// TwinCAT 3 PLC project IBF_HMI
// Title: IBF_HMI
// Company: Industrial Brains B.V.
// ProjectVersion: 0.0.0.0
// Description: Basic HMI screens for use with Utilities and device libraries
// ProgramVersion: 3.1.4023.0
// libraries:
//   IBF_Devices, * (Industrial Brains B.V.)
//   IBF_Utilities, * (Industrial Brains B.V.)
//   Tc2_Standard, * (Beckhoff Automation GmbH)
//   Tc2_System, * (Beckhoff Automation GmbH)
//   Tc2_Utilities, * (Beckhoff Automation GmbH)
//   Tc3_Module, * (Beckhoff Automation GmbH)
//   VisuDialogs, * (System)
//   VisuSymbols,3.5.10.0,System
// project tree:
//   HMIControl/DataTypes/ E_BaseVisu.TcTLEO, UDT_HMI_FaultLogItem.TcDUT, UDT_HMI_LogItem.TcDUT
//   HMIControl/ FB_LogView.TcPOU, FB_HMIControl.TcPOU
//   IconsAndPictures/Backgrounds/ BackgroundImagePool_PNG.TcIPO (not stored), BackGroundImagePool_SVG.TcIPO (not stored)
//   / PlcTask.TcTTO, VisualizationManager.TcVMO (not stored), VISU_TASK.TcTTO
//   Screens/Backgrounds/ BG_Borders.TcVIS, BG_Emergency.TcVIS, BG_Logo_IndustrialBrains.TcVIS
//   Screens/Base/ BaseScreen.TcVIS
//   Screens/Buttons/ ButtonHome.TcVIS, ButtonLogin.TcVIS, ButtonManual.TcVIS, ButtonSettings.TcVIS, ButtonParameters.TcVIS, ButtonLog.TcVIS, ButtonTemplate.TcVIS
//   Screens/LogView/ LogView.TcVIS
//   Screens/Parameter/ ParameterControl.TcVIS
//   Screens/State/ Idle.TcVIS, Manual.TcVIS, Parameters.TcVIS, FaultLog.TcVIS
//   Tools/Colors/ E_Color.TcDUT, F_GetColor.TcPOU, F_GetTransparantColor.TcPOU, U_Color.TcDUT
//   Tools/InputFunctions/ FB_HMIInputBase.TcPOU, FB_HMILREALInput.TcPOU
//   _TESTS/ FB_Base_Test.TcPOU, PRG_TEST.TcPOU, PRG_TEST_GLOBAL.TcPOU, PRG_TEST_LOGVIEW.TcPOU, VISU_DummyState.TcVIS, VISU_TEST_BASE.TcVIS, VISU_TEST_LOGVIEW.TcVIS
//   GVL/ GVL_HMI.TcGVL
//   IconsAndPictures/Buttons/ Buttons_SVG.TcIPO (not stored), Buttons_PNG.TcIPO (not stored)
//   IconsAndPictures/Logos/ LogoPool.TcIPO (not stored)
//   TextLists/ E_ComponentTypes.TcTLO, E_FaultTypes.TcTLO (not stored), E_Locations.TcTLO (not stored), E_MessageNumbers.TcTLO, E_ParameterNames.TcTLO (not stored), GlobalTextList.TcGTLO, TL_MessageDiscriptions.TcTLO (not stored)
// real-time tasks:
//   TASK PlcTask: cycle T#10ms, priority 6, ADS port 350
//   TASK VISU_TASK: cycle T#100000us, priority 8, ADS port 351

CONFIGURATION IBF_HMI
    RESOURCE PLC ON TwinCAT3
        TASK PlcTask(INTERVAL := T#10ms, PRIORITY := 6);
        TASK VISU_TASK(INTERVAL := T#100000us, PRIORITY := 8);
        PROGRAM PRG_TEST_GLOBAL WITH PlcTask : PRG_TEST_GLOBAL;
        PROGRAM PRG_TEST WITH PlcTask : PRG_TEST;
        PROGRAM PRG_TEST_LOGVIEW WITH PlcTask : PRG_TEST_LOGVIEW;
        PROGRAM VisuElems_Visu_Prg WITH VISU_TASK : VisuElems.Visu_Prg;
    END_RESOURCE
END_CONFIGURATION

// ---- HMIControl/DataTypes/E_BaseVisu.TcTLEO
{attribute 'qualified_only'}
{attribute 'strict'}
TYPE E_BaseVisu :
(
	Idle := 0,
	Settings,
	Parameter,
	Manual,
	SemiAutomatic,
	Automatic,
	LogView
)INT;
END_TYPE

// ---- HMIControl/DataTypes/UDT_HMI_FaultLogItem.TcDUT
TYPE UDT_HMI_FaultLogItem :
STRUCT
	sID : STRING;
	sDescription : STRING;
	sStartTime : STRING[19];
	sEndTime : STRING[19];
	dColor_Bg : DWORD := E_Color.White; // Table row background color
END_STRUCT
END_TYPE

// ---- HMIControl/DataTypes/UDT_HMI_LogItem.TcDUT
TYPE UDT_HMI_LogItem :
STRUCT
	sTimestamp : STRING[23];
	sLevel : STRING;
	sMsg : T_MaxString;
	dColor_Bg : DWORD := E_Color.White; // Table row background color
END_STRUCT
END_TYPE

// ---- Tools/Colors/E_Color.TcDUT
{attribute 'qualified_only'}
{attribute 'strict'}
TYPE E_Color : // Theme colors
(
	Bg_Light	:= 16#FF19A9E1, // Theme background color (light blue)
	Bg_Dark		:= 16#FF122941, // Theme background color (dark blue)

	White 		:= 16#FFFFFFFF,
	Black 		:= 16#FF000000,

	DarkRed		:= 16#FFFF0000,
	LightRed	:= 16#FFFF8888,
	DarkYellow 	:= 16#FFFFFF00,
	LightYellow := 16#FFFFFF88,
	DarkGreen 	:= 16#FF00FF00,
	LightGreen	:= 16#FF88FF88

) DWORD;
END_TYPE

// ---- Tools/Colors/U_Color.TcDUT
TYPE U_Color :
UNION
	rgba : ARRAY[0..3] OF BYTE;
	dw : DWORD;
END_UNION
END_TYPE

// ---- GVL/GVL_HMI.TcGVL
{attribute 'qualified_only'}
VAR_GLOBAL
	fbHMIControl	: FB_HMIControl ; // HMI control function
END_VAR

// ---- _TESTS/PRG_TEST_GLOBAL.TcPOU
PROGRAM INTERNAL PRG_TEST_GLOBAL // A place to call global function blocks (singletons) that can be used by all tests

Sys_Variables.fbSystemVariables();
GVL_Utilities.fbFaultHandler();

END_PROGRAM

// ---- _TESTS/PRG_TEST.TcPOU
PROGRAM INTERNAL PRG_TEST
VAR
	fbLogHandler_PersistentArray : FB_LogHandler_PersistentArray;
	bInitDone 	: BOOL;
	fbDevValve 	: FB_DevValve;
END_VAR

// NOTE: fbParameterHandler should contain the parameters of fbDevValve. 
// Parameter values are persistent
IF NOT bInitDone THEN
	bInitDone := TRUE;
	fbDevValve.Init(
		nId := 1,
		nParentId := 0,
		eResetState := E_ValveResetState.Res_Idle,
		eSafeState := E_ValveResetState.Res_Idle
	);
END_IF

fbDevValve();

GVL_Parameters.fbParameterHandler();

GVL_HMI.fbHMIControl(fbLogHandler_PersistentArray := fbLogHandler_PersistentArray);

END_PROGRAM

// ---- _TESTS/PRG_TEST_LOGVIEW.TcPOU
PROGRAM INTERNAL PRG_TEST_LOGVIEW
VAR
	fbLogHandler_PersistentArray : FB_LogHandler_PersistentArray;
	bEnableTests : BOOL;
	fbLogView : FB_LogView;
	fbLogger : FB_Logger;
	fbBase : FB_Base_Test;
	bCmdReset : BOOL;
END_VAR

IF bEnableTests THEN

	fbLogView(fbLogHandler_PersistentArray := fbLogHandler_PersistentArray);

	fbBase();

	IF bCmdReset THEN
		bCmdReset R= GVL_Utilities.fbFaultHandler.CmdReset();
	END_IF
	
END_IF

END_PROGRAM

// ---- HMIControl/FB_LogView.TcPOU
FUNCTION_BLOCK INTERNAL FB_LogView
VAR CONSTANT
	NUMBER_OF_ITEMS_IN_TABLE : UINT := 16;
END_VAR
VAR_INPUT
	bAcknowledge : BOOL; // Clear inactive items from the log
	bReset : BOOL; // Reset faults
	bBlinkButton : BOOL; // Blink the button to alert operator (optional, not used thusfar)
	fbLogHandler_RetainableList : REFERENCE TO FB_LogHandler_RetainableList; // Optional reference to a FB_LogHandler_RetainableList instance
END_VAR
VAR_OUTPUT
	arLog : ARRAY[1..NUMBER_OF_ITEMS_IN_TABLE] OF UDT_HMI_FaultLogItem;
	arHistory : ARRAY[1..GVL_Utilities.RETAINABLE_LOG_HISTORY_SIZE] OF UDT_HMI_LogItem;
	
	// Log button properties
	dLogButtonColor 	: DWORD;
	nLogButtonNumber 	: UINT;
		
	reNewLogMessages : BOOL; // TRUE when new log messages arrive (for one cycle)
	nPrevFaultsInLog : UINT;
END_VAR
VAR
	fbFormatString : FB_FormatString;
END_VAR
VAR_TEMP
	i : UINT; // Iterator
	nArHistoryIndex : UINT; // arHistory array index
	
	stLogItem : UDT_LogItem;
	stFaultLogItem : UDT_FaultLogItem;
	stEmptyFaultLogItem : UDT_HMI_FaultLogItem;
	
	fMonth : REAL;
	fDay : REAL;
	fHour : REAL;
	fMinute : REAL;
	fSecond : REAL;
	fMilliseconds : REAL;	
END_VAR

{region 'FAULT LOG / ALARM BELL ICON'}
// Report new log messages
reNewLogMessages := (GVL_Utilities.fbFaultHandler.nFaultsInLog > nPrevFaultsInLog);
nPrevFaultsInLog := GVL_Utilities.fbFaultHandler.nFaultsInLog;

// Update array
stFaultLogItem := GVL_Utilities.fbFaultHandler.Head;
FOR i := 1 TO NUMBER_OF_ITEMS_IN_TABLE DO
	IF i <= GVL_Utilities.fbFaultHandler.nFaultsInLog THEN
		arLog[i].sID := stFaultLogItem.Id;
		arLog[i].sDescription := stFaultLogItem.stFault.Description;
		arLog[i].sStartTime := DT_To_Str(stFaultLogItem.StartTime);
		arLog[i].sEndTime := DT_To_Str(stFaultLogItem.EndTime);
		IF stFaultLogItem.stFault.Active THEN
			arLog[i].dColor_Bg := GetFaultTypeColorBG(stFaultLogItem.stFault.FaultType);
		ELSE
			arLog[i].dColor_Bg := E_Color.White;
		END_IF
		stFaultLogItem := GVL_Utilities.fbFaultHandler.Next;
	ELSE
		arLog[i] := stEmptyFaultLogItem;
	END_IF
END_FOR

// Set log button properties
nLogButtonNumber := GVL_Utilities.fbFaultHandler.nFaultsInLog;
// Set color, in order of priority
IF bBlinkButton AND Sys_Variables.BlinkFast THEN
	dLogButtonColor := E_Color.Bg_Dark;
ELSIF GVL_Utilities.fbFaultHandler.arActiveFaultTypes[E_FaultTypes.FF] THEN
	dLogButtonColor := GetFaultTypeColorBG(E_FaultTypes.FF);
ELSIF GVL_Utilities.fbFaultHandler.arActiveFaultTypes[E_FaultTypes.CF] THEN
	dLogButtonColor := GetFaultTypeColorBG(E_FaultTypes.CF);
ELSIF GVL_Utilities.fbFaultHandler.arActiveFaultTypes[E_FaultTypes.MC] THEN
	dLogButtonColor := GetFaultTypeColorBG(E_FaultTypes.MC);
ELSIF GVL_Utilities.fbFaultHandler.arActiveFaultTypes[E_FaultTypes.OW] THEN
	dLogButtonColor := GetFaultTypeColorBG(E_FaultTypes.OW);
ELSIF GVL_Utilities.fbFaultHandler.arActiveFaultTypes[E_FaultTypes.OM] THEN
	dLogButtonColor := GetFaultTypeColorBG(E_FaultTypes.OM);
ELSE
	dLogButtonColor := E_Color.Bg_Light;
END_IF 

IF bAcknowledge THEN
	bAcknowledge R= GVL_Utilities.fbFaultHandler.CmdClearInactive();
END_IF

IF bReset THEN
	bReset R= GVL_Utilities.fbFaultHandler.CmdReset();
END_IF
{endregion}

{region 'Log history'}
IF __ISVALIDREF(fbLogHandler_RetainableList) THEN
	// Add items from retainable list in reversed order, starting with the last added item
	nArHistoryIndex := 0;
	FOR i := (fbLogHandler_RetainableList.nIndex + GVL_Utilities.RETAINABLE_LOG_HISTORY_SIZE - 1) TO fbLogHandler_RetainableList.nIndex BY -1 DO
		nArHistoryIndex := nArHistoryIndex + 1;
		stLogItem := fbLogHandler_RetainableList.aLogItems[(i MOD GVL_Utilities.RETAINABLE_LOG_HISTORY_SIZE) + 1];
		arHistory[nArHistoryIndex].sMsg := TO_STRING(stLogItem.sMsg);
		arHistory[nArHistoryIndex].sLevel := TO_STRING(stLogItem.eLevel);
		arHistory[nArHistoryIndex].dColor_Bg := GetLevelColorBG(stLogItem.eLevel);

		// Build timestamp string
		fMonth := WORD_TO_REAL(stLogItem.stTimestamp.wMonth); 
		fDay := WORD_TO_REAL(stLogItem.stTimestamp.wDay); 
		fHour := WORD_TO_REAL(stLogItem.stTimestamp.wHour); 
		fMinute := WORD_TO_REAL(stLogItem.stTimestamp.wMinute); 
		fSecond := WORD_TO_REAL(stLogItem.stTimestamp.wSecond); 
		fMilliseconds := WORD_TO_REAL(stLogItem.stTimestamp.wMilliseconds);
		fbFormatString(
			sFormat := '%u-%02.0f-%02.0f %02.0f:%02.0f:%02.0f.%03.0f',
			arg1 := F_WORD(stLogItem.stTimestamp.wYear),
			arg2 := F_REAL(fMonth),
			arg3 := F_REAL(fDay),
			arg4 := F_REAL(fHour),
			arg5 := F_REAL(fMinute),
			arg6 := F_REAL(fSecond),
			arg7 := F_REAL(fMilliseconds),
			sOut => arHistory[nArHistoryIndex].sTimestamp
		);
	END_FOR
END_IF
{endregion}

METHOD PRIVATE GetFaultTypeColorBG : DWORD
VAR_INPUT
	eFaultType : E_FaultTypes;
END_VAR
CASE eFaultType OF
	E_FaultTypes.FF:
		GetFaultTypeColorBG := E_Color.LightRed;
	E_FaultTypes.CF:
		GetFaultTypeColorBG := E_Color.LightRed;
	E_FaultTypes.MC:
		GetFaultTypeColorBG := E_Color.LightYellow;
	E_FaultTypes.OW:
		GetFaultTypeColorBG := E_Color.LightYellow;
	E_FaultTypes.OM:
		GetFaultTypeColorBG := E_Color.Bg_Light;
END_CASE
END_METHOD

METHOD PRIVATE GetLevelColorBG : DWORD
VAR_INPUT
	eLogLevel : E_LogLevel;
END_VAR
CASE eLogLevel OF
	E_LogLevel.TRACE:
		GetLevelColorBG := E_Color.White;
	E_LogLevel.DEBUG:
		GetLevelColorBG := E_Color.White;
	E_LogLevel.INFO:
		GetLevelColorBG := E_Color.LightGreen;
	E_LogLevel.WARN:
		GetLevelColorBG := E_Color.LightYellow;
	E_LogLevel.ERROR:
		GetLevelColorBG := E_Color.LightRed;
	E_LogLevel.FATAL:
		GetLevelColorBG := E_Color.LightRed;
END_CASE
END_METHOD

END_FUNCTION_BLOCK

// ---- _TESTS/FB_Base_Test.TcPOU
FUNCTION_BLOCK INTERNAL FB_Base_Test EXTENDS FB_Base

SUPER^();

METHOD PUBLIC Init : BOOL
VAR_INPUT
	nId				: UINT ; // Identification number of object
	nParentId		: UINT ; // Id of higher level if applicable (0 = no parent)
	eComponentType	: E_ComponentTypes ; // Component or function type
END_VAR
// Every FB_Base instance is expected to have an Init method that calls ExecIdentifyDevice. 
// This Init method will have at least the nId and nParentId inputs.
// The eComponentType input is optional (can be hardcoded in the Init method, for example see FB_Step).
// It might also have additional inputs (changing the method signature) therefore it is not declared in FB_Base.
ExecIdentifyDevice(nId,	nParentId,	eComponentType);
END_METHOD

END_FUNCTION_BLOCK

// ---- HMIControl/FB_HMIControl.TcPOU
FUNCTION_BLOCK FB_HMIControl
VAR_INPUT
	eScreenRequest 			: E_BaseVisu;
	eHomeScreen   			: E_BaseVisu := E_BaseVisu.Idle; // Home screen is based on system state, e.g., Idle, Automatic, etc.

	bShowEmergencyOverlay 	: BOOL;
	sEmergencyText 			: STRING; // Visible when emergency overlay is shown
	sStatusText 			: STRING; // Text in the bottom border of the screen 

	fbLogHandler_RetainableList : REFERENCE TO FB_LogHandler_RetainableList; // Optional reference to a FB_LogHandler_RetainableList instance
END_VAR
VAR_OUTPUT
	eShownScreen : E_BaseVisu := E_BaseVisu.Idle;

	// Screen states
	bInScreenHome 		: BOOL;
	bInScreenSettings 	: BOOL;
	bInScreenManual 	: BOOL;
	bInScreenParameters	: BOOL;
	bInScreenLog		: BOOL;
	
	// Hide admin/service level navigation buttons
	bHideSecureButtons : BOOL;
END_VAR
VAR
	fbLogView			: FB_LogView;

	feWriteParameter 	: F_TRIG ; // Falling edge trigger on leaving parameter or manual screen
	bWritePar  			: BOOL ; // Busy writing parameters
END_VAR

// Run log view handler
fbLogView(fbLogHandler_RetainableList := fbLogHandler_RetainableList);

// Check user level
bHideSecureButtons := NOT (VisuElems.CurrentUserGroupName = "Admin" OR VisuElems.CurrentUserGroupName = "Service");

// Check if logged in user is allowed to be in the current screen. If not, go to home screen.
IF bHideSecureButtons AND ((eShownScreen = E_BaseVisu.Manual) OR (eShownScreen = E_BaseVisu.Parameter)) THEN
	eScreenRequest := E_BaseVisu.Idle;
END_IF 

// Switch screen
IF (eScreenRequest = E_BaseVisu.Idle) THEN
	eShownScreen := eHomeScreen;
ELSIF (eScreenRequest <> eShownScreen) THEN
	eShownScreen := eScreenRequest;
END_IF

// Report screen states
bInScreenHome 		:= (eShownScreen = eHomeScreen); 
bInScreenSettings 	:= (eShownScreen = E_BaseVisu.Settings);
bInScreenManual 	:= (eShownScreen = E_BaseVisu.Manual);
bInScreenLog 		:= (eShownScreen = E_BaseVisu.LogView);
bInScreenParameters := (eShownScreen = E_BaseVisu.Parameter);

// Save parameters after leaving parameter of manual screen
// Note: in manual operation one can change parameters as well ("learn" function)
feWriteParameter(CLK := (eShownScreen = E_BaseVisu.Parameter) OR (eShownScreen = E_BaseVisu.Manual));
IF feWriteParameter.Q THEN
	bWritePar := TRUE;
END_IF
IF bWritePar THEN 
	bWritePar R= GVL_Parameters.fbParameterHandler.CmdSavePar();
END_IF

END_FUNCTION_BLOCK

// ---- Tools/Colors/F_GetColor.TcPOU
FUNCTION F_GetColor : DWORD // Return an opaque color in DWORD format for use in visualisation
VAR_INPUT
	Red : BYTE;
	Green : BYTE;
	Blue : BYTE;
END_VAR
VAR
END_VAR

F_GetColor := F_GetTransparantColor(Red, Green, Blue, 16#FF);

END_FUNCTION

// ---- Tools/Colors/F_GetTransparantColor.TcPOU
FUNCTION F_GetTransparantColor : DWORD  // Return a transparant color in DWORD format for use in visualisation
VAR_INPUT
	Red : BYTE;
	Green : BYTE;
	Blue : BYTE;
	Alpha : BYTE := 16#FF; // Transparancy, 0 = fully transparant
END_VAR
VAR
	uColor : U_Color;
END_VAR

uColor.rgba[0] := Red;
uColor.rgba[1] := Green;
uColor.rgba[2] := Blue;
uColor.rgba[3] := Alpha;
F_GetTransparantColor := uColor.dw;

END_FUNCTION

// ---- Tools/InputFunctions/FB_HMIInputBase.TcPOU
FUNCTION_BLOCK ABSTRACT FB_HMIInputBase //Base function for HMI inputs
VAR_INPUT
	bEnable : BOOL := TRUE ;
END_VAR
VAR_OUTPUT
	bInVisible			: BOOL := TRUE ; // input is visible (standard := NOT bEnable )
	bDeactivateInput	: BOOL := TRUE ; // input is enabled (Standard := bEnable)
END_VAR
VAR
END_VAR

SetHMIInstructions();

METHOD INTERNAL SetHMIInstructions : BOOL
VAR_INPUT
END_VAR
bInVisible 			:= NOT bEnable ;
bDeactivateInput	:= NOT bEnable ;
END_METHOD

METHOD ABSTRACT SetOutputToPLC : BOOL
VAR_INPUT
END_VAR
END_METHOD

END_FUNCTION_BLOCK

// ---- Tools/InputFunctions/FB_HMILREALInput.TcPOU
FUNCTION_BLOCK PUBLIC FB_HMILREALInput EXTENDS FB_HMIInputBase // Analog value input from HMI
VAR_INPUT
	fInputFromHMI	: LREAL ;
END_VAR
VAR_OUTPUT
	fOutputToPLC	: LREAL ;
END_VAR
VAR
END_VAR

// call base function 
SUPER^();

// Set output to PLC
SetOutputToPLC();

METHOD PUBLIC SetOutputToPLC : BOOL
VAR_INPUT
END_VAR
IF bEnable THEN 
	fOutputToPLC := fInputFromHMI ;
END_IF
END_METHOD

END_FUNCTION_BLOCK

// ---- Screens/Backgrounds/BG_Borders.TcVIS
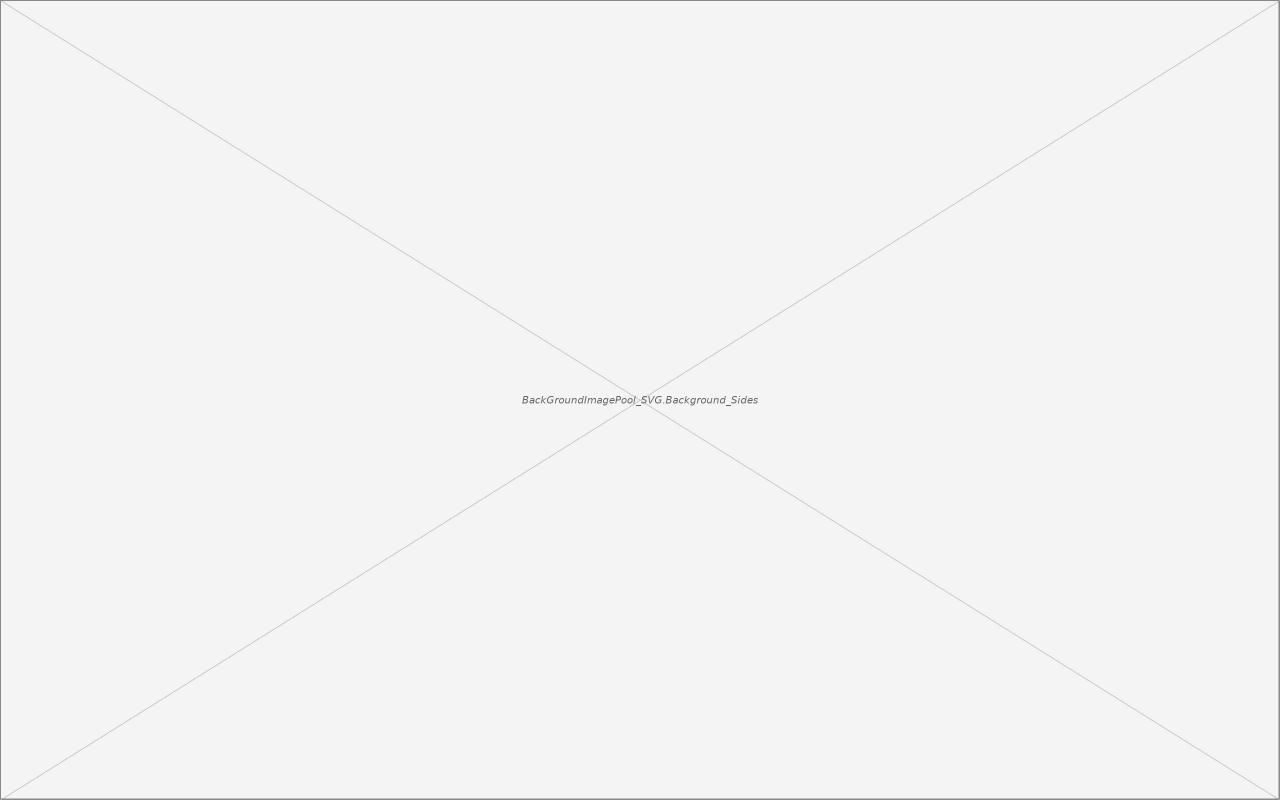
VISUALIZATION BG_Borders  // 1280x800
    Image (0,710 1280x90), image: BackGroundImagePool_SVG.Background_Bottom
    Image (0,0 1280x800), image: BackGroundImagePool_SVG.Background_Sides
END_VISUALIZATION

// ---- Screens/Backgrounds/BG_Emergency.TcVIS
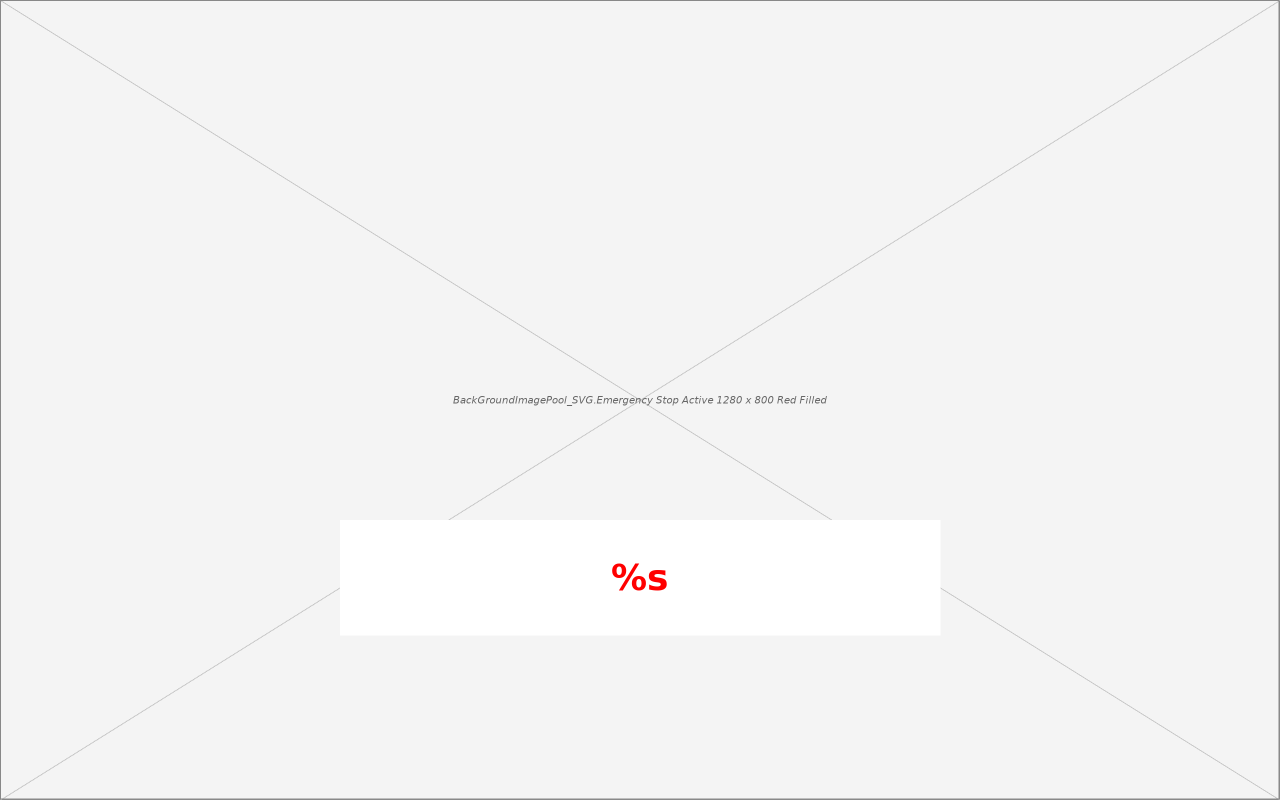
VISUALIZATION BG_Emergency  // 1280x800
VAR_IN_OUT
	sMessage : STRING;
END_VAR
    Image (0,0 1280x800), invisible if: NOT GVL_HMI.fbHMIControl.bShowEmergencyOverlay, image: BackGroundImagePool_SVG.Emergency Stop Active 1280 x 800 Red Filled
    Textfield (340,520 600x115), "%s", text variable: sMessage
END_VISUALIZATION

// ---- Screens/Backgrounds/BG_Logo_IndustrialBrains.TcVIS
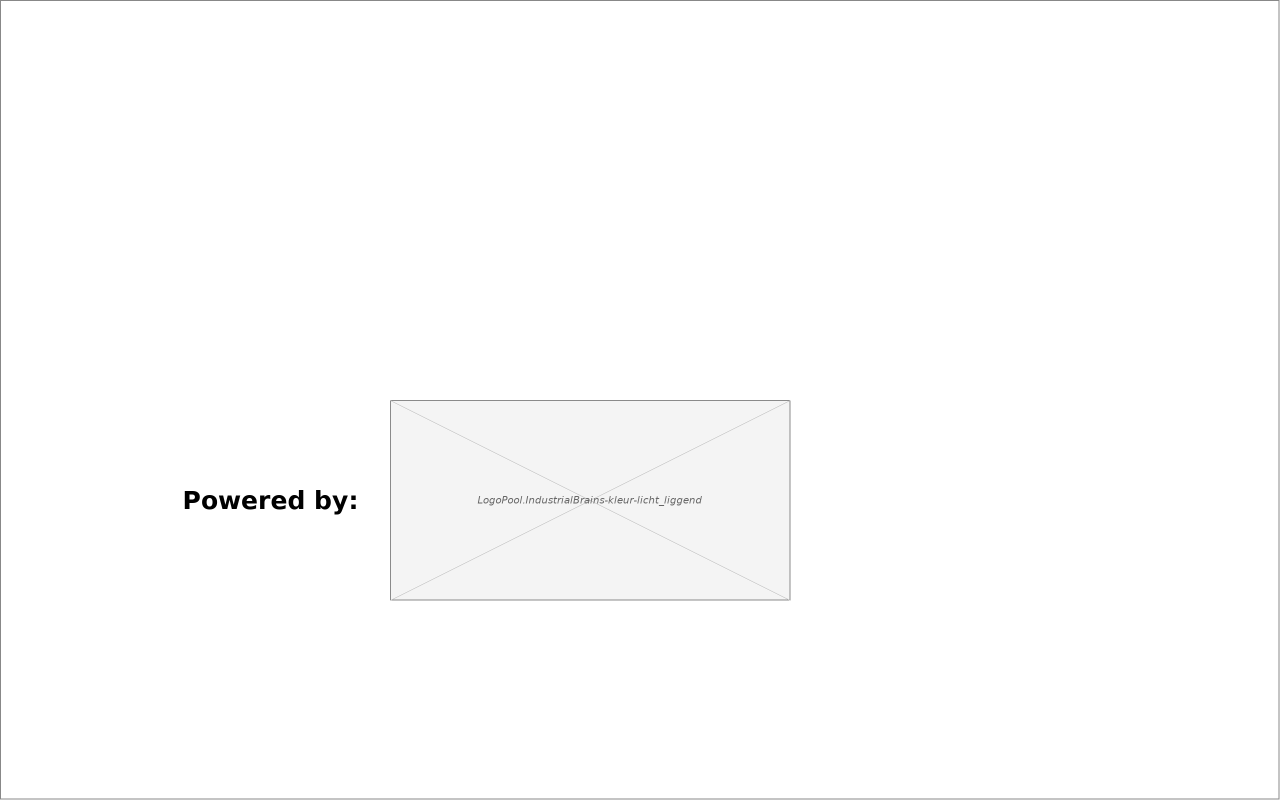
VISUALIZATION BG_Logo_IndustrialBrains  // 1280x800
    Image (390,400 400x200), image: LogoPool.IndustrialBrains-kleur-licht_liggend
    Label (170,400 200x200), "Powered by:"
END_VISUALIZATION

// ---- Screens/Base/BaseScreen.TcVIS
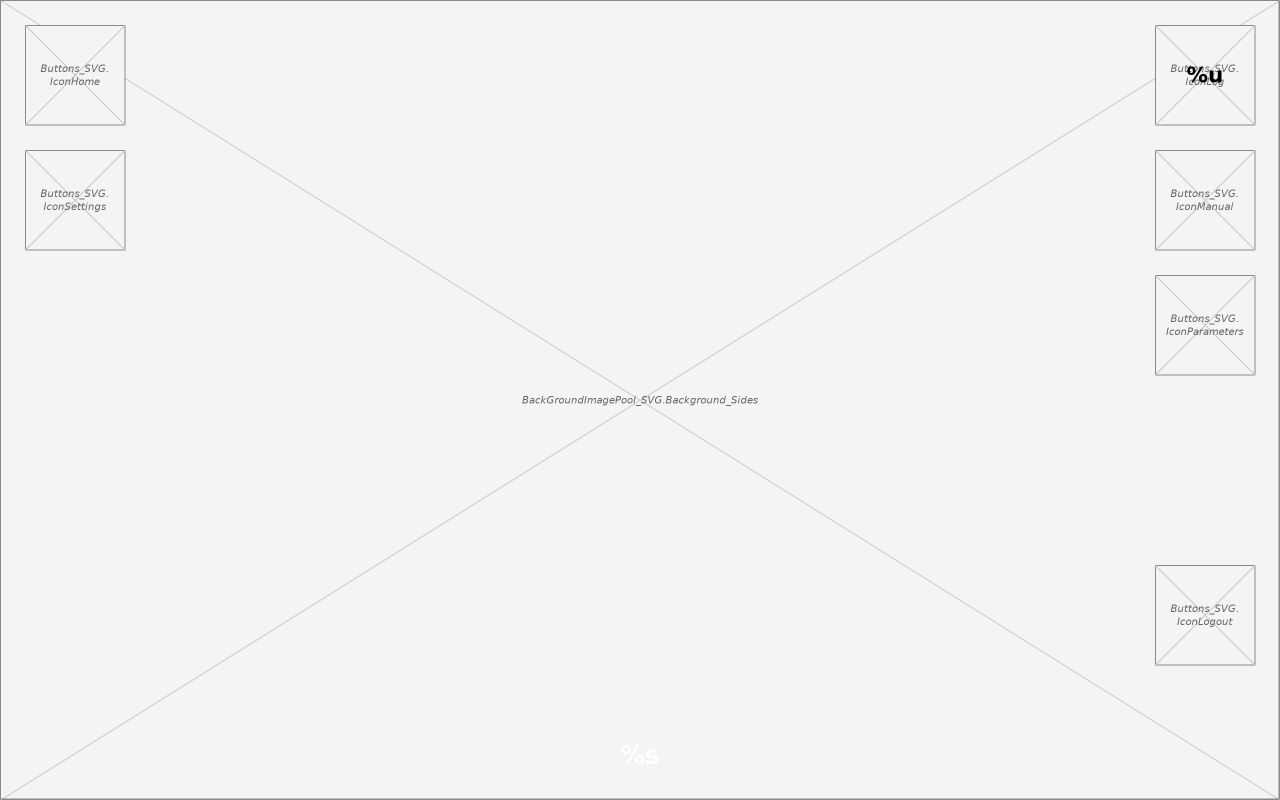
VISUALIZATION BaseScreen  // 1280x800
    Frame (0,0 1280x800)
        shows BG_Borders()
    Frame (25,25 100x100)
        shows ButtonHome(bState := GVL_HMI.fbHMIControl.bInScreenHome)
    Frame (25,150 100x100)
        shows ButtonSettings(bState := GVL_HMI.fbHMIControl.bInScreenSettings)
    Frame (1155,150 100x100), invisible if: GVL_HMI.fbHMIControl.bHideSecureButtons
        shows ButtonManual(bState := GVL_HMI.fbHMIControl.bInScreenManual)
    Frame (1155,275 100x100), invisible if: GVL_HMI.fbHMIControl.bHideSecureButtons
        shows ButtonParameters(bState := GVL_HMI.fbHMIControl.bInScreenParameters)
    Frame (1155,25 100x100)
        shows ButtonLog(bState := GVL_HMI.fbHMIControl.bInScreenLog, nNumber := GVL_HMI.fbHMIControl.fbLogView.nLogButtonNumber, dColor := GVL_HMI.fbHMIControl.fbLogView.dLogButtonColor)
    Frame (1155,565 100x100)
        shows ButtonLogin()
    Textfield (550,730 180x50), "%s", text variable: GVL_HMI.fbHMIControl.sStatusText
END_VISUALIZATION

// ---- Screens/Buttons/ButtonHome.TcVIS
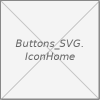
VISUALIZATION ButtonHome  // 100x100
VAR_IN_OUT
	bState : BOOL;
END_VAR
    Frame (0,0 100x100)
        shows ButtonTemplate(bActive := bState)
    Image (0,0 100x100), image: Buttons_SVG.IconHome
        OnMouseDown: execute { GVL_HMI.fbHMIControl.eScreenRequest := E_BaseVisu.Idle; }
END_VISUALIZATION

// ---- Screens/Buttons/ButtonLogin.TcVIS
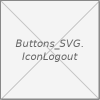
VISUALIZATION ButtonLogin  // 100x100
    Ellipse (0,0 100x100)
    Image (0,0 100x100), image: Buttons_SVG.IconLogin
        OnMouseDown: VisuUserMgmt Type=Login
    Ellipse (0,0 100x100)
    Image (0,0 100x100), image: Buttons_SVG.IconLogout
        OnMouseDown: VisuUserMgmt Type=Logout
END_VISUALIZATION

// ---- Screens/Buttons/ButtonManual.TcVIS
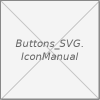
VISUALIZATION ButtonManual  // 100x100
VAR_IN_OUT
	bState : BOOL;
END_VAR
    Frame (0,0 100x100)
        shows ButtonTemplate(bActive := bState)
    Image (0,0 100x100), image: Buttons_SVG.IconManual
        OnMouseDown: execute { GVL_HMI.fbHMIControl.eScreenRequest := E_BaseVisu.Manual; }
END_VISUALIZATION

// ---- Screens/Buttons/ButtonSettings.TcVIS
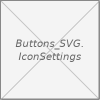
VISUALIZATION ButtonSettings  // 100x100
VAR_IN_OUT
	bState : BOOL;
END_VAR
    Frame (0,0 100x100)
        shows ButtonTemplate(bActive := bState)
    Image (0,0 100x100), image: Buttons_SVG.IconSettings
        OnMouseDown: execute { GVL_HMI.fbHMIControl.eScreenRequest := E_BaseVisu.Settings; }
END_VISUALIZATION

// ---- Screens/Buttons/ButtonParameters.TcVIS
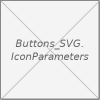
VISUALIZATION ButtonParameters  // 100x100
VAR_IN_OUT
	bState : BOOL;
END_VAR
    Frame (0,0 100x100)
        shows ButtonTemplate(bActive := bState)
    Image (0,0 100x100), image: Buttons_SVG.IconParameters
        OnMouseDown: execute { GVL_HMI.fbHMIControl.eScreenRequest := E_BaseVisu.Parameter; }
END_VISUALIZATION

// ---- Screens/Buttons/ButtonLog.TcVIS
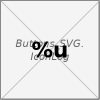
VISUALIZATION ButtonLog  // 100x100
VAR_IN_OUT
	bState : BOOL;
	nNumber : UINT;
	dColor : DWORD;
END_VAR
    Frame (0,0 100x100)
        shows ButtonTemplate(bActive := bState)
    Ellipse (5,5 90x90), colour variable: dColor
    Image (0,0 100x100), image: Buttons_SVG.IconLog
    Textfield (0,0 100x100), "%u", text variable: nNumber
        OnMouseDown: execute { GVL_HMI.fbHMIControl.eScreenRequest := E_BaseVisu.LogView; }
END_VISUALIZATION

// ---- Screens/Buttons/ButtonTemplate.TcVIS
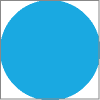
VISUALIZATION ButtonTemplate  // 100x100
VAR_IN_OUT
	bActive : BOOL;	
END_VAR
    Ellipse (0,0 100x100), colour toggle: bActive
    Ellipse (5,5 90x90)
END_VISUALIZATION

// ---- Screens/LogView/LogView.TcVIS
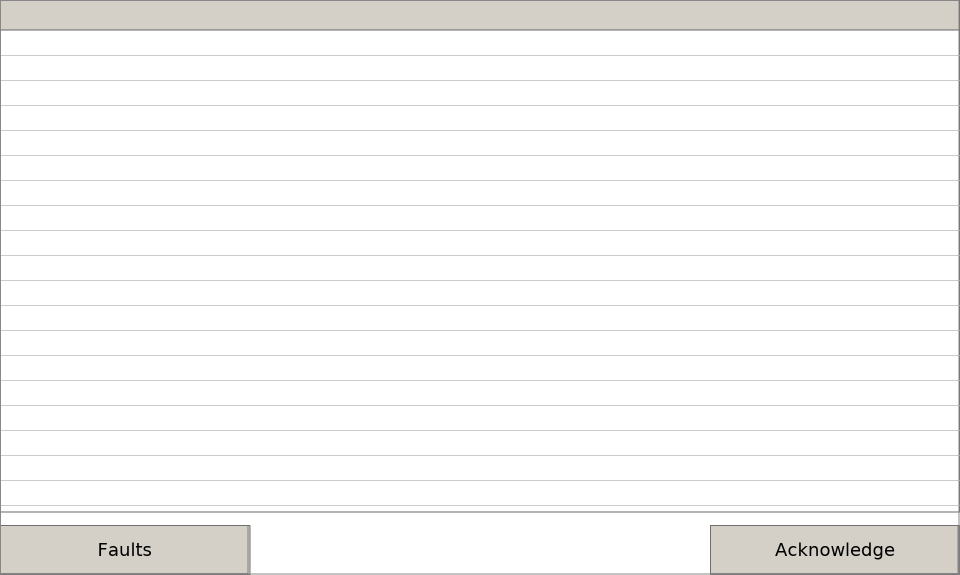
VISUALIZATION LogView  // 960x575
VAR_IN_OUT
	// NOTE: LogView table rows should match IBF_Utilities library parameter PAR_Utilities.MAX_FAULTS_IN_LOG
	fbLogView : FB_LogView;
END_VAR
VAR
	bShowLogHistory : BOOL; // Show the log history instead of the fault list
END_VAR
    Table (0,0 960x512), invisible if: bShowLogHistory, data array: fbLogView.arLog
        p3854506369: fbLogView.arLog[INDEX].sID
        p1892666644: fbLogView.arLog [INDEX].sDescription
        p338671338: fbLogView.arLog [INDEX].sStartTime
        p2170511999: fbLogView.arLog [INDEX].sEndTime
        p3723444502: fbLogView.arLog [INDEX].dColor_Bg
        p2685023577: fbLogView.arLog [INDEX].sID
        Columns.Column.[0].Template: fbLogView.arLog[INDEX].dColor_Bg
        Columns.Column.[1].Template: fbLogView.arLog[INDEX].dColor_Bg
        Columns.Column.[2].Template: fbLogView.arLog[INDEX].dColor_Bg
        Columns.Column.[3].Template: fbLogView.arLog[INDEX].dColor_Bg
    Table (0,0 960x512), invisible if: NOT bShowLogHistory, data array: fbLogView.arHistory
        p3723444502: fbLogView.arLog [INDEX].dColor_Bg
        p3854506369: fbLogView.arHistory[INDEX].sTimestamp
        p1892666644: fbLogView.arHistory[INDEX].sLevel
        p338671338: fbLogView.arHistory[INDEX].sMsg
        p2170511999: fbLogView.arHistory[INDEX].dColor_Bg
        p1755163831: Message
        Columns.Column.[3].Template: fbLogView.arLog[INDEX].dColor_Bg
    Button (710,525 250x50), "Acknowledge"
        tap fbLogView.bAcknowledge
    Button (0,525 250x50), "History", invisible if: bShowLogHistory
        toggle bShowLogHistory
    Button (0,525 250x50), "Faults", invisible if: NOT bShowLogHistory
        toggle bShowLogHistory
END_VISUALIZATION

// ---- Screens/Parameter/ParameterControl.TcVIS
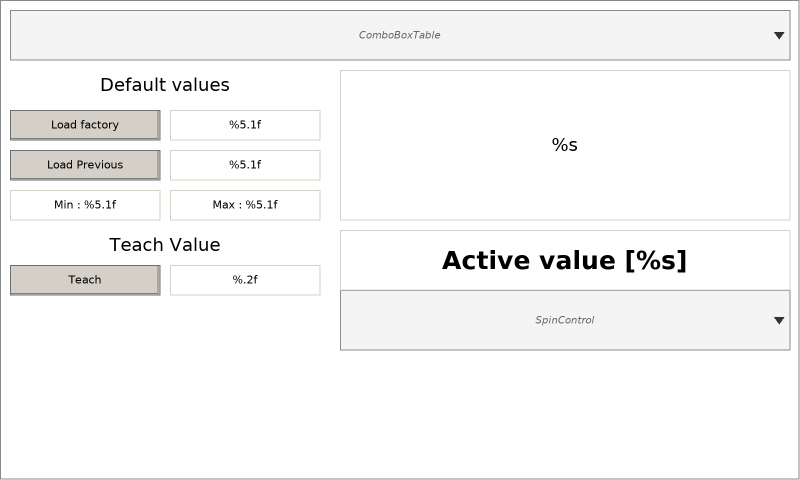
VISUALIZATION ParameterControl  // 800x480
    ComboBoxTable (10,10 780x50), variable: GVL_Parameters.fbParameterHandler.nLookupIndex, data array: GVL_Parameters.fbParameterHandler.arParameters
        p1128707560: GVL_Parameters.fbParameterHandler.nNumberOfParameters
        p3854506369: GVL_Parameters.fbParameterHandler.arParameters[INDEX].nNumber
        p1892666644: GVL_Parameters.fbParameterHandler.arParameters[INDEX].sName
        p338671338: GVL_Parameters.fbParameterHandler.arParameters[INDEX].sType
        p2170511999: GVL_Parameters.fbParameterHandler.arParameters[INDEX].pParameter^
    Group (10,70 310x150)
        Button (0,40 150x30), "Load factory"
            tap GVL_Parameters.fbParameterHandler.bCmdLoadfactory
        Label (0,0 310x30), "Default values"
        Textfield (160,40 150x30), "%5.1f", text variable: GVL_Parameters.fbParameterHandler.arParameters[GVL_Parameters.fbParameterHandler.nLookupIndex].pParameter^.fFactory
            OnMouseClick: write the text variable via VisuDialogs.Numpad, min GVL_Parameters.fbParameterHandler.arParameters[GVL_Parameters.fbParameterHandler.nLookupIndex].pParameter^.fMinimum, max GVL_Parameters.fbParameterHandler.arParameters[GVL_Parameters.fbParameterHandler.nLookupIndex].pParameter^.fMaximum
        Button (0,80 150x30), "Load Previous"
            tap GVL_Parameters.fbParameterHandler.bCmdLoadFromPrevious
        Textfield (160,80 150x30), "%5.1f", text variable: GVL_Parameters.fbParameterHandler.arParameters[GVL_Parameters.fbParameterHandler.nLookupIndex].pParameter^.fSaved
        Textfield (160,120 150x30), "Max : %5.1f", text variable: GVL_Parameters.fbParameterHandler.arParameters[GVL_Parameters.fbParameterHandler.nLookupIndex].pParameter^.fMaximum
            OnMouseClick: write the text variable via VisuDialogs.Numpad
        Textfield (0,120 150x30), "Min : %5.1f", text variable: GVL_Parameters.fbParameterHandler.arParameters[GVL_Parameters.fbParameterHandler.nLookupIndex].pParameter^.fMinimum
            OnMouseClick: write the text variable via VisuDialogs.Numpad
    Textfield (340,70 450x150), "%s", text variable: GVL_Parameters.fbParameterHandler.arParameters[GVL_Parameters.fbParameterHandler.nLookupIndex].pParameter^.sDiscription
    SpinControl (340,290 450x60), variable: GVL_Parameters.fbParameterHandler.arParameters[GVL_Parameters.fbParameterHandler.nLookupIndex].pParameter^.fValue
        p576042468: GVL_Parameters.fbParameterHandler.arParameters[GVL_Parameters.fbParameterHandler.nLookupIndex].pParameter^.fMinimum
        p651134158: GVL_Parameters.fbParameterHandler.arParameters[GVL_Parameters.fbParameterHandler.nLookupIndex].pParameter^.fMaximum
        OnMouseClick: write the text variable via VisuDialogs.Numpad, min GVL_Parameters.fbParameterHandler.arParameters[GVL_Parameters.fbParameterHandler.nLookupIndex].pParameter^.fMinimum, max GVL_Parameters.fbParameterHandler.arParameters[GVL_Parameters.fbParameterHandler.nLookupIndex].pParameter^.fMaximum
    Textfield (340,230 450x60), "Active value [%s]", text variable: GVL_Parameters.fbParameterHandler.arParameters[GVL_Parameters.fbParameterHandler.nLookupIndex].pParameter^.sUnit
    Group (10,230 310x65)
        Label (0,0 310x30), "Teach Value"
        Textfield (160,35 150x30), "%.2f", text variable: GVL_Parameters.fbParameterHandler.arParameters[GVL_Parameters.fbParameterHandler.nLookupIndex].pParameter^.fPrepared
        Button (0,35 150x30), "Teach"
            tap GVL_Parameters.fbParameterHandler.bCmdAcceptTeach
END_VISUALIZATION

// ---- Screens/State/Idle.TcVIS
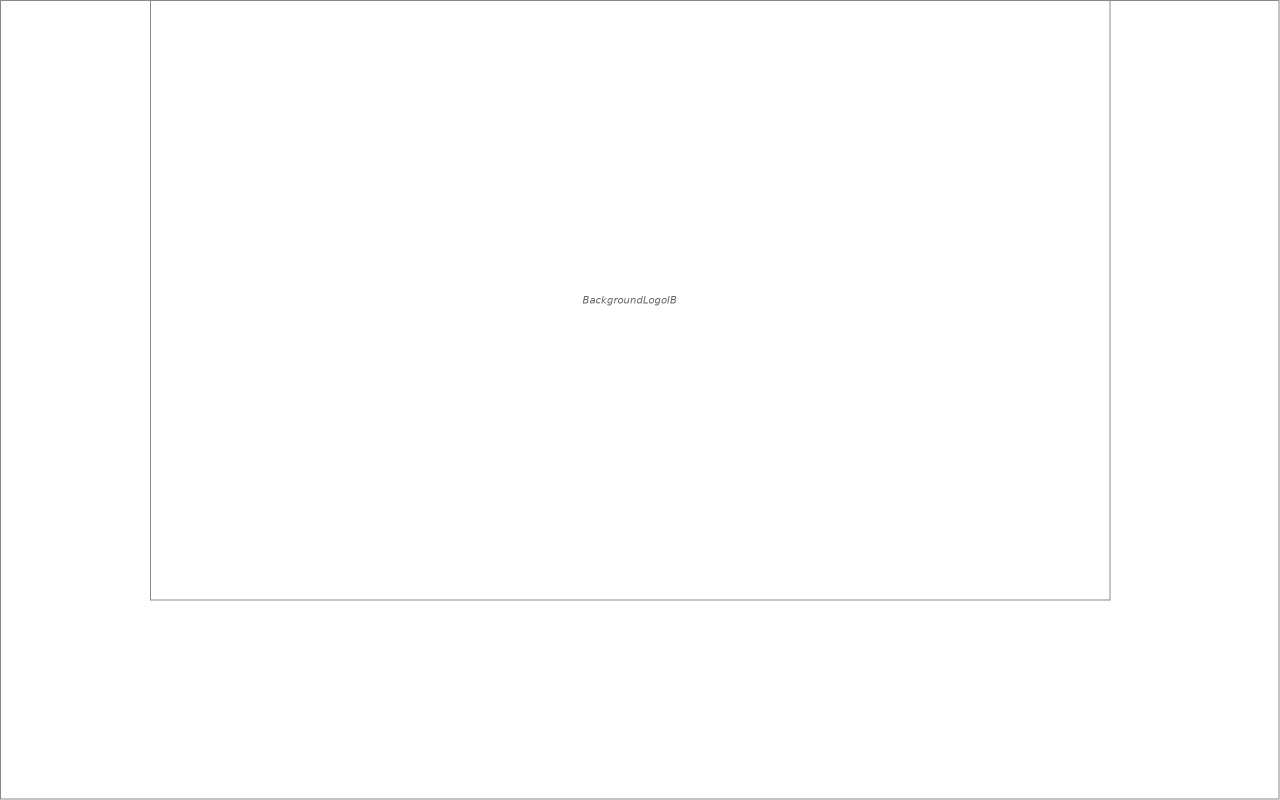
VISUALIZATION Idle  // 1280x800
    Frame (150,0 960x600)
        shows BackgroundLogoIB()
END_VISUALIZATION

// ---- Screens/State/Manual.TcVIS
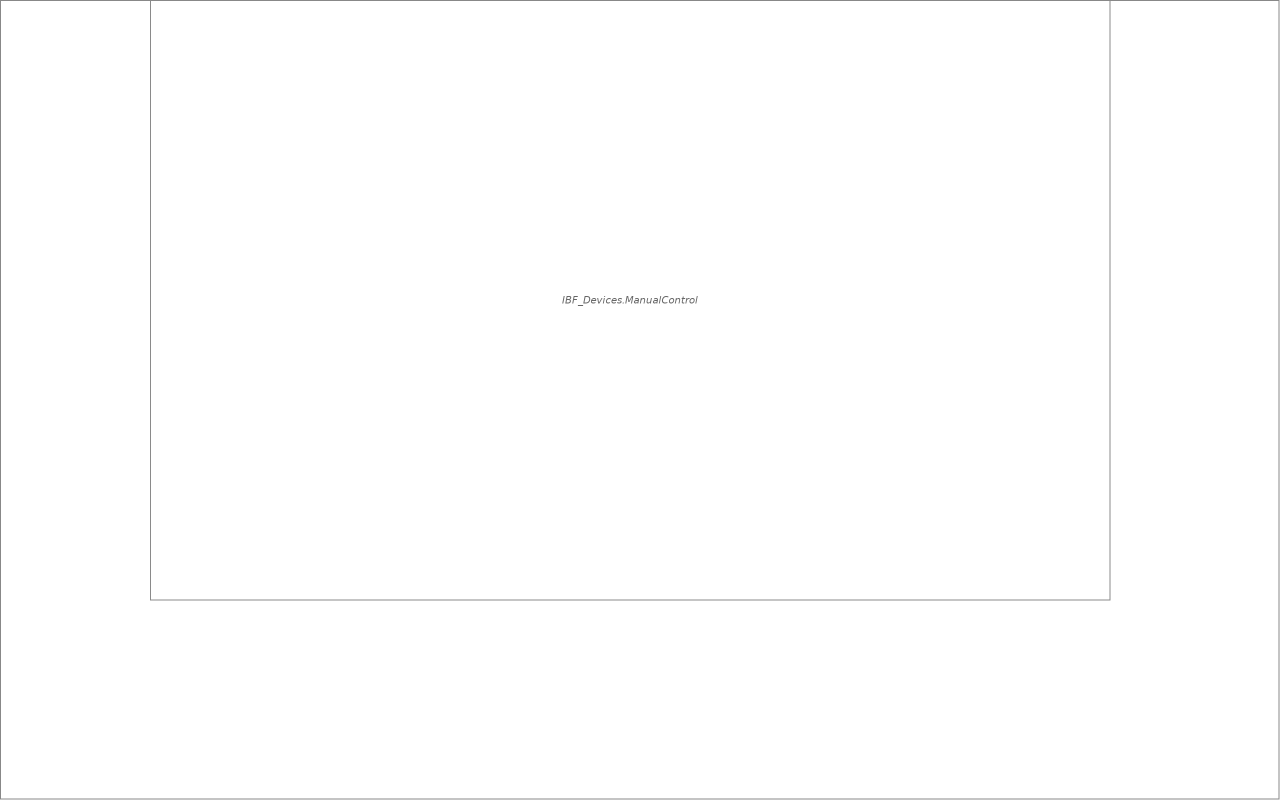
VISUALIZATION Manual  // 1280x800
    Frame (150,0 960x600)
        shows IBF_Devices.ManualControl(stHMI := GVL_Devices.fbManualController.stHMI, fbManualController := GVL_Devices.fbManualController)
END_VISUALIZATION

// ---- Screens/State/Parameters.TcVIS
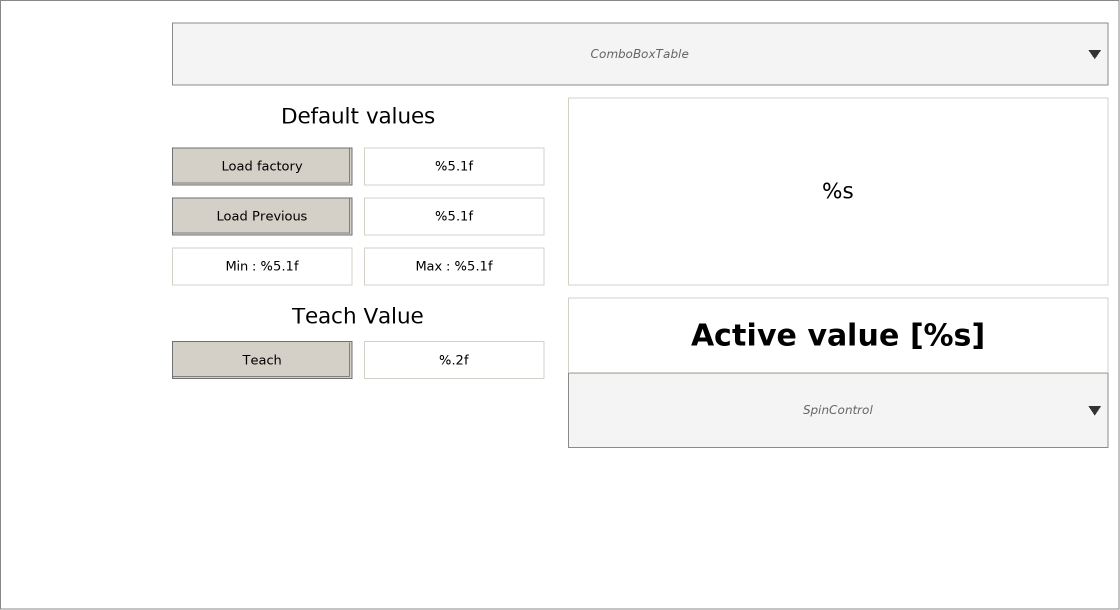
VISUALIZATION Parameters  // 1120x610
    Frame (160,10 960x600)
        shows ParameterControl()
END_VISUALIZATION

// ---- Screens/State/FaultLog.TcVIS
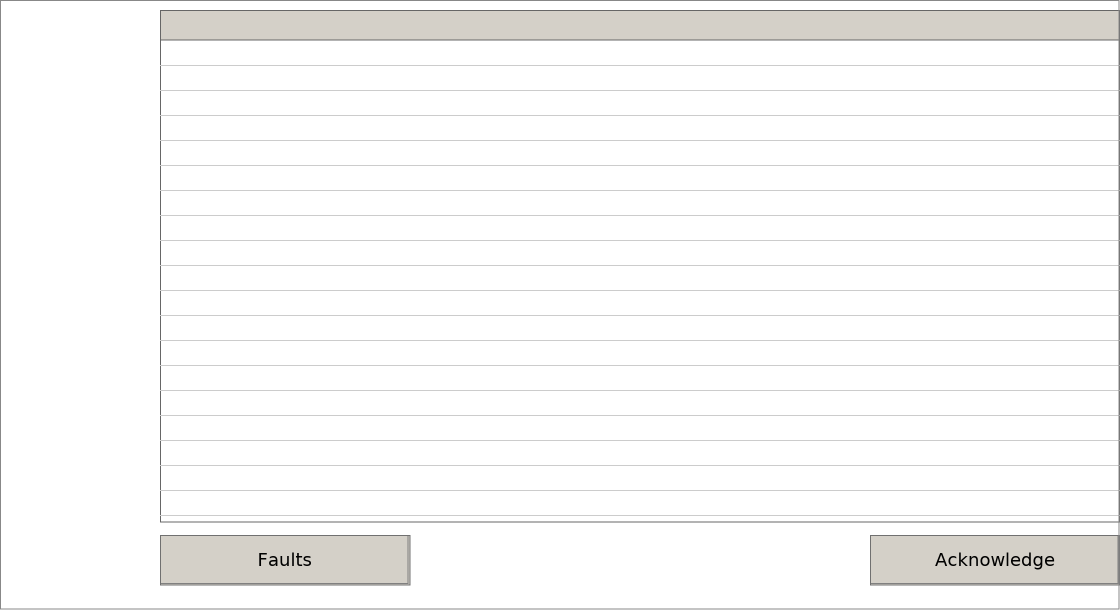
VISUALIZATION FaultLog  // 1120x610
VAR_IN_OUT
	fbLogger : FB_Logger;
END_VAR
    Frame (160,10 960x600)
        shows LogView(fbLogView := GVL_HMI.fbHMIControl.fbLogView)
END_VISUALIZATION

// ---- _TESTS/VISU_DummyState.TcVIS
VISUALIZATION VISU_DummyState  // 2x2
END_VISUALIZATION

// ---- _TESTS/VISU_TEST_BASE.TcVIS
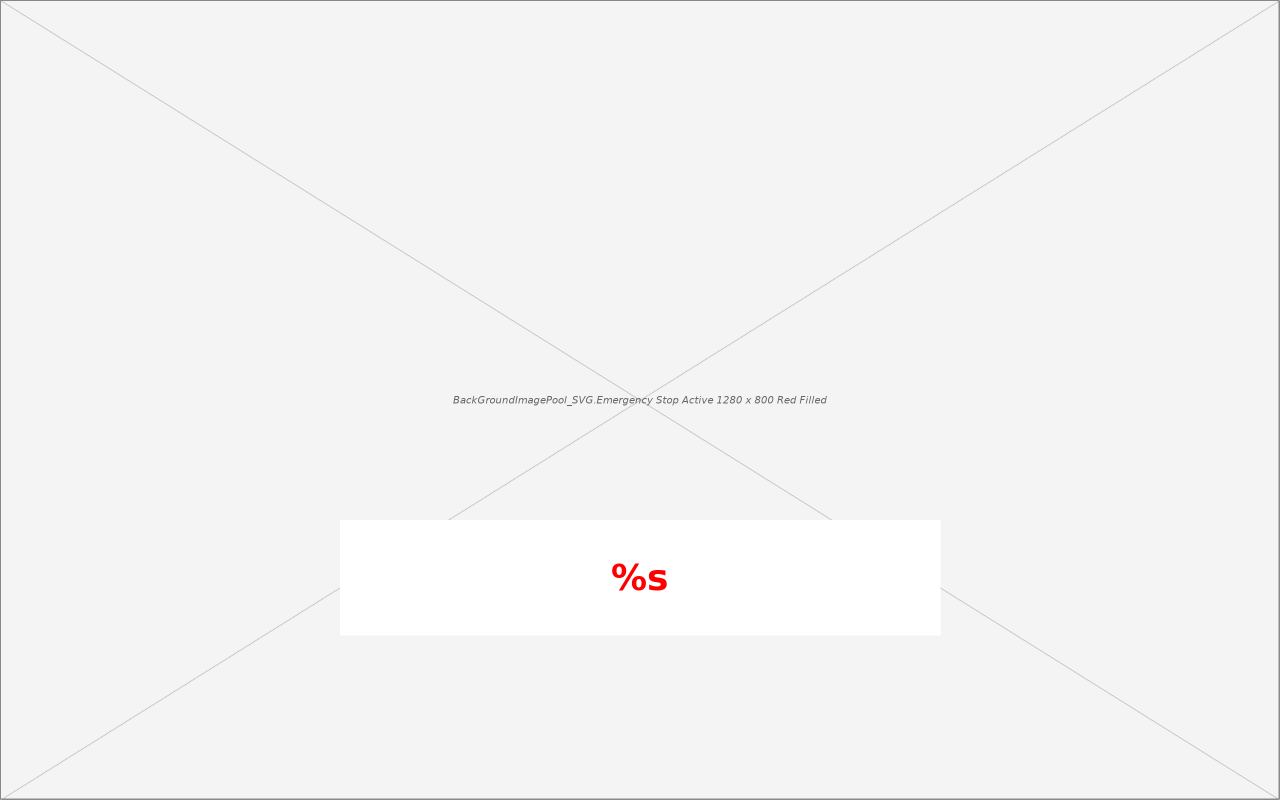
VISUALIZATION VISU_TEST_BASE  // 1280x800
    Frame (0,0 1280x800)
        shows BaseScreen()
    Frame (0,0 1280x800), frame switch variable: GVL_HMI.fbHMIControl.eShownScreen
        shows Idle()
        shows VISU_DummyState()
        shows Parameters()
        shows Manual()
        shows VISU_DummyState()
        shows VISU_DummyState()
        shows FaultLog(fbLogger := PRG_TEST_LOGVIEW.fbLogger)
    Frame (0,0 1280x800), invisible if: NOT GVL_HMI.fbHMIControl.bShowEmergencyOverlay
        shows BG_Emergency(sMessage := GVL_HMI.fbHMIControl.sEmergencyText)
END_VISUALIZATION

// ---- _TESTS/VISU_TEST_LOGVIEW.TcVIS
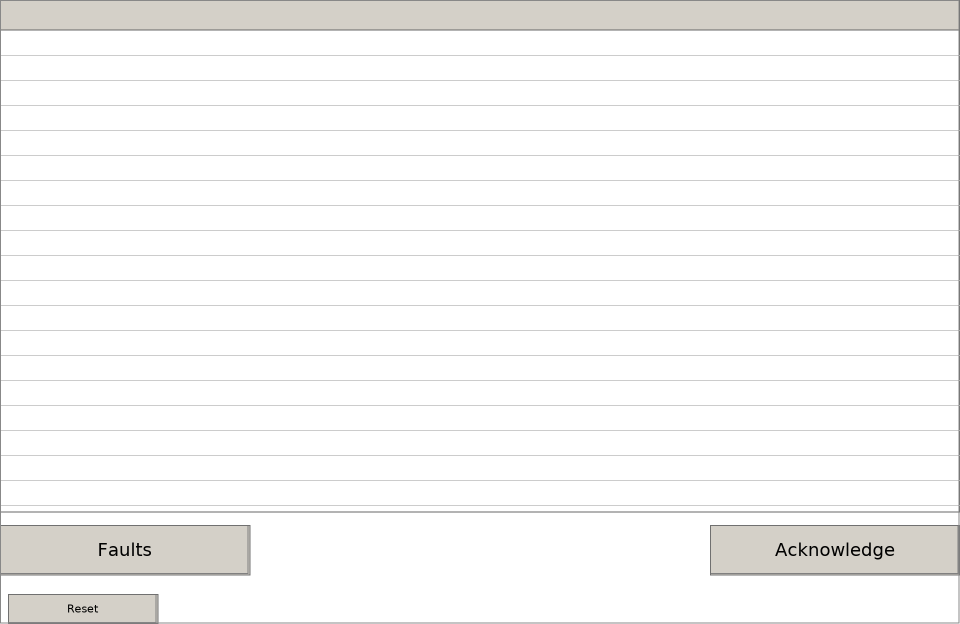
VISUALIZATION VISU_TEST_LOGVIEW  // 960x624
    Frame (0,0 960x512)
        shows LogView(fbLogView := PRG_TEST_LOGVIEW.fbLogView)
    Button (8,594 150x30), "Reset"
        tap PRG_TEST_LOGVIEW.fbLogView.bReset
END_VISUALIZATION

// ---- TextLists/E_ComponentTypes.TcTLO
TEXTLIST E_ComponentTypes
  0 = 'NA'
  10 = 'Cylinder'
  11 = 'Axis'
  20 = 'EstopButton'
  21 = 'EstopBumper'
  22 = 'Pushbutton'
  23 = 'Switch'
  30 = 'SafeIO'
  31 = 'Rio_Box'
  32 = 'Rio_Slot'
  33 = 'Encoder'
  34 = 'DiSensor'
  40 = 'ServoDrive'
  50 = 'HMI'
  51 = 'RemoteOS'
  52 = 'RemoteDB'
  60 = 'Assembly'
  61 = 'SubAssembly'
  100 = 'MainProgram'
  101 = 'StepProgram'
  102 = 'FunctionBlock'
   = ''
END_TEXTLIST

// ---- TextLists/E_MessageNumbers.TcTLO
TEXTLIST E_MessageNumbers
  0 = 'NA_NoMessage'
  1 = 'FF_Unknown'
  2 = 'FF_NoCommunication'
  3 = 'FF_ComunicationFault'
  4 = 'FF_Overload'
  5 = 'FF_EncoderFault'
  6 = 'FF_SlaveFault'
  7 = 'FF_AxisFault'
  8 = 'FF_DriveFault'
  9 = 'FF_Collision'
  100 = 'CF_FeedbackFault'
  101 = 'CF_WrongDirection'
  102 = 'CF_MoveToFast'
  103 = 'CF_MoveToSlow'
  104 = 'CF_WrongPosition'
  105 = 'CF_Obstruction'
  200 = 'MC_WaitingForproduct'
  201 = 'MC_WaitingForOperator'
  202 = 'MC_WaitingForModule'
  203 = 'MC_WaitingForMaster'
  204 = 'MC_WaitingForSlave'
  205 = 'MC_WrongPosition'
  300 = 'OM_AlmostEmpty'
  301 = 'OM_Finished'
  302 = 'OM_ready'
  900 = 'FF_MessageTest'
  901 = 'CF_MessageTest'
  902 = 'MC_MessageTest'
  903 = 'OM_MessageTest'
   = ''
END_TEXTLIST

// ---- TextLists/GlobalTextList.TcGTLO
TEXTLIST GlobalTextList
  268 = '%.2f'
  923 = '%5.1f'
  596 = '%s'
  689 = '%u'
  352 = 'Acknowledge'
  638 = 'Active value [%s]'
  1038 = 'Admin'
  264 = 'Default values'
  1228 = 'Faults'
  344 = 'History'
  291 = 'Level'
  154 = 'Load factory'
  624 = 'Load Previous'
  133 = 'Log'
  278 = 'Max : %5.1f'
  269 = 'Message'
  520 = 'Min : %5.1f'
  298 = 'None'
  293 = 'Operator'
  482 = 'Powered by: '
  174 = 'Reset'
  284 = 'Service'
  771 = 'Teach'
  229 = 'Teach Value'
  10 = 'Timestamp'
END_TEXTLIST
